FUNCTION_BLOCK FB_SoftWash IMPLEMENTS I_WashStrategy
VAR
     stWashSettings   : ST_WashSettings;
     bStarted   : BOOL := FALSE;
END_VAR

METHOD FB_init : BOOL
VAR_INPUT
	bInitRetains : BOOL; // if TRUE, the retain variables are initialized (warm start / cold start)
	bInCopyCode : BOOL;  // if TRUE, the instance afterwards gets moved into the copy code (online change)
END_VAR
stWashSettings.tFillDuration  := GVL_WashConstants.SOFT_FILL;
stWashSettings.tWashDuration  := GVL_WashConstants.SOFT_WASH;
stWashSettings.tDrainDuration := GVL_WashConstants.SOFT_DRAIN;
stWashSettings.rWashTemperature   := GVL_WashConstants.SOFT_TEMP;
stWashSettings.nSpinSpeed     := GVL_WashConstants.SOFT_SPEED;
stWashSettings.sDescription   := 'Soft wash — gentle cycle low temp';

FB_init := TRUE;
END_METHOD

{warning 'add method implementation '}
METHOD GetDuration : TIME
GetDuration := stWashSettings.tWashDuration;
END_METHOD

{warning 'add method implementation '}
METHOD GetProgramName : STRING
GetProgramName := 'SOFT WASH';
END_METHOD

{warning 'add method implementation '}
METHOD GetWashSettings : ST_WashSettings
GetWashSettings := stWashSettings;
END_METHOD

{warning 'add method implementation '}
METHOD Start : BOOL
bStarted := TRUE;
Start     := TRUE;
END_METHOD

END_FUNCTION_BLOCK

(* stored: Version 1.1.0.1, ProductVersion 3.1.4024.16
   POU FB_SoftWash: Id {6b043722-bfdb-4fc2-b930-ac005af82bce}, SpecialFunc None
   Method FB_init: Id {ac107336-e5fd-4103-89a4-917f149c10b4}
   Method GetDuration: Id {f79856c6-80e5-4073-b33b-b6aa5da6a2ed}
   Method GetProgramName: Id {e19bdd1e-d922-44db-b6c0-a2a741b58381}
   Method GetWashSettings: Id {df66c8da-2696-4042-ac99-05daf904a1d9}
   Method Start: Id {93c3279d-abbc-40ce-a312-81023cabebf8} *)
